Staubli VAL3: Step1.dtx

mdesc mNomSpeed
pointRx Starting_point = {x=-380, y=80, z=150, rx=180, rz=-90, fatherId=world[0]}
pointRx Real_start = {fatherId=world[0]}
pointRx B = {rx=180, fatherId=world[0]}
pointRx C = {rx=180, fatherId=world[0]}
pointRx D = {rx=180, fatherId=world[0]}
pointRx E = {rx=180, fatherId=world[0]}
num Dim_width
num Dim_height
screen sEcran
num nYN
num nx
num ny
num nz
num nRx
num nRy
num nRz
tool tTool = {fatherId=flange[0], ioLink=valve1}
pointRx pCentrepiece1[4]
  [0] = {x=-170, y=-290, rx=180, rz=-90, fatherId=world[0]}
  [1] = {x=-56, y=-290, rx=180, rz=-90, fatherId=world[0]}
  [2] = {x=58, y=-290, rx=180, rz=-90, fatherId=world[0]}
  [3] = {x=170, y=-290, rx=180, rz=-90, fatherId=world[0]}
num nNbPieceMax = 6
num nNbPieceArrive
pointRx Real_Stop = {fatherId=world[0]}
pointRx pCentre_Arrive[7]
  [0] = {y=335, rx=180, fatherId=world[0]}
  [1] = {y=240, rx=180, fatherId=world[0]}
  [2] = {x=50, y=290, rx=180, rz=90, fatherId=world[0]}
  [3] = {x=-50, y=290, rx=180, rz=90, fatherId=world[0]}
  [4] = {x=-20, y=290, rx=180, rz=90, fatherId=world[0]}
  [5] = {x=20, y=290, rx=180, rz=90, fatherId=world[0]}
  [6] = {y=290, z=150, rx=180, fatherId=world[0]}
pointRx pTestTemp = {y=-290, z=-180, rx=180, fatherId=world[0]}
pointRx B_haut = {fatherId=world[0]}
num i
num nNbEtage
num DepotStock[4]
  [0] = 5
  [1] = 5
  [2] = 5
  [3] = 5
num indiceStock
num nValeurAngle
